FUNCTION_BLOCK FB_NOTT_ZNSE_ACTUATORS
VAR_INPUT
END_VAR
VAR_OUTPUT
END_VAR
VAR
	NGP1:		FB_NOTT_MOTOR;
	NGP2:		FB_NOTT_MOTOR;
	NGP3:		FB_NOTT_MOTOR;
	NGP4:		FB_NOTT_MOTOR;
	
	
	ptrNGPs:	ARRAY [1..4] OF POINTER TO FB_NOTT_MOTOR;
	// GUI stuff
	guiNGPsIndex:	UINT := 1;	// Index for Shutter Engineering GUI
	
	stat:		T_NOTT_STAT;
	
END_VAR



NGP1(
	in_bSafe:=, 
	in_bDisableIfUnsafe:=, 
	sName:= 'NDL1', 
	nNOVRAM_DevId:= 6, 
	nNOVRAM_Offset:= 29000);
	
NGP2(
	in_bSafe:=, 
	in_bDisableIfUnsafe:=, 
	sName:= 'NDL2', 
	nNOVRAM_DevId:= 6, 
	nNOVRAM_Offset:= 30000);
	
NGP3(
	in_bSafe:=, 
	in_bDisableIfUnsafe:=, 
	sName:= 'NDL3', 
	nNOVRAM_DevId:= 6, 
	nNOVRAM_Offset:= 31000);
	
NGP4(
	in_bSafe:=, 
	in_bDisableIfUnsafe:=, 
	sName:= 'NDL4', 
	nNOVRAM_DevId:= 6, 
	nNOVRAM_Offset:= 32000);

	
M_Configure();

METHOD M_Configure : BOOL
VAR_INPUT
END_VAR

ptrNGPs[1] := ADR(NGP1);
ptrNGPs[2] := ADR(NGP2);
ptrNGPs[3] := ADR(NGP3);
ptrNGPs[4] := ADR(NGP4);
END_METHOD

END_FUNCTION_BLOCK

(* stored: Version 1.1.0.1, ProductVersion 3.1.4024.14
   POU FB_NOTT_ZNSE_ACTUATORS: Id {9528e71d-9f9f-4df0-98bb-0baeaffdac59}, SpecialFunc None
   Method M_Configure: Id {e4ab5b72-2f0f-428a-aaf4-51528fb78fc8} *)
